// TIA Portal V17 export
// export: Created 2023-02-14T02:49:46.4601409Z, ExportSetting WithDefaults, DisplayName Totally Integrated Automation Portal, DisplayVersion V17, DisplayName TIA Portal Openness, DisplayVersion V17, DisplayName TIA Portal Teamcenter Gateway, DisplayVersion V17, DisplayName TIA Portal Version Control Interface, DisplayVersion V17, DisplayName SINAMICS Startdrive Advanced, DisplayVersion V17, DisplayName SINAMICS Startdrive G130, G150, S120, S150, SINAMICS MV, S210, DisplayVersion V17, DisplayName SINAMICS Startdrive G110M, G120, G120C, G120D, G120P, G115D, DisplayVersion V17, DisplayName STEP 7 Professional, DisplayVersion V17, DisplayName STEP 7 Safety, DisplayVersion V17, DisplayName WinCC Professional, DisplayVersion V17
FUNCTION "IO Homoge" : Void   // FC1, LAD
{ S7_Optimized_Access := 'TRUE' }
VERSION : 0.1
// stored: AutoNumber true, IsIECCheckEnabled false, SetENOAutomatically false, UDAEnableTagReadback false
BEGIN

REGION Network 1: Analog
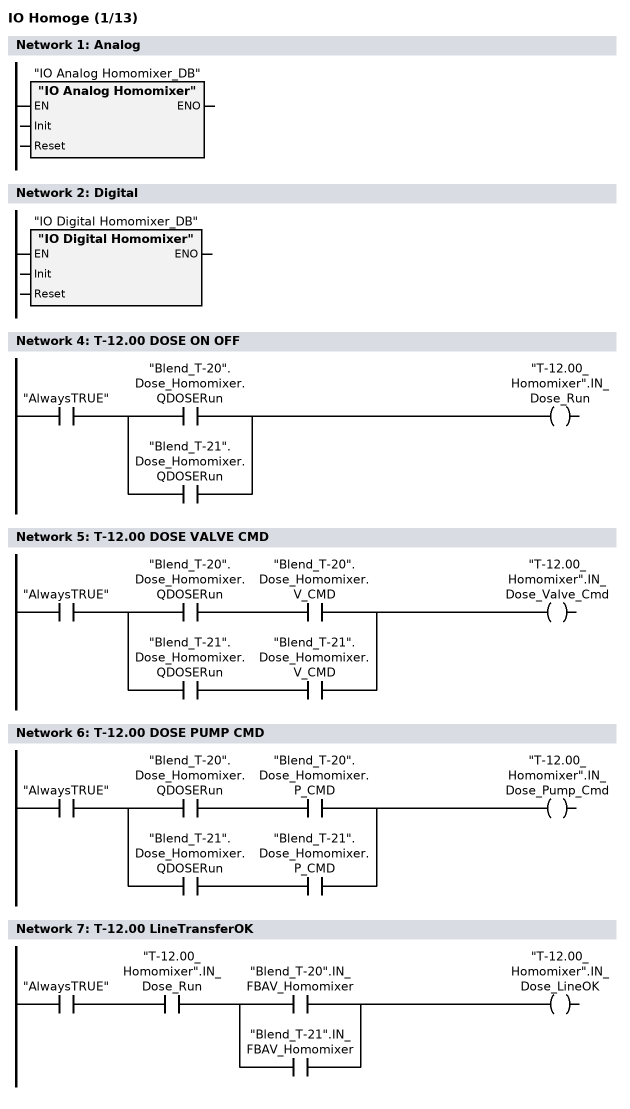
   RUNG wire#powerrail
      "IO Analog Homomixer_DB"(Init :=, Reset :=)
   END_RUNG
   // the same network as SCL:
   "IO Analog Homomixer_DB"();   // "IO Analog Homomixer"
END_REGION

REGION Network 2: Digital
   RUNG wire#powerrail
      "IO Digital Homomixer_DB"(Init :=, Reset :=)
   END_RUNG
   // the same network as SCL:
   "IO Digital Homomixer_DB"();   // "IO Digital Homomixer"
END_REGION

REGION Network 4: T-12.00 DOSE ON OFF
   RUNG wire#powerrail
      Contact( "AlwaysTRUE" )
      wire#w1
      Contact( "Blend_T-20".Dose_Homomixer.QDOSERun )
      wire#w2
      Coil( "T-12.00_Homomixer".IN_Dose_Run )
   END_RUNG
   RUNG wire#w1
      Contact( "Blend_T-21".Dose_Homomixer.QDOSERun )
   END_RUNG wire#w2
   // the same network as SCL:
   "T-12.00_Homomixer".IN_Dose_Run := "AlwaysTRUE" AND ("Blend_T-20".Dose_Homomixer.QDOSERun OR "Blend_T-21".Dose_Homomixer.QDOSERun);
END_REGION

REGION Network 5: T-12.00 DOSE VALVE CMD
   RUNG wire#powerrail
      Contact( "AlwaysTRUE" )
      wire#w1
      Contact( "Blend_T-20".Dose_Homomixer.QDOSERun )
      Contact( "Blend_T-20".Dose_Homomixer.V_CMD )
      wire#w2
      Coil( "T-12.00_Homomixer".IN_Dose_Valve_Cmd )
   END_RUNG
   RUNG wire#w1
      Contact( "Blend_T-21".Dose_Homomixer.QDOSERun )
      Contact( "Blend_T-21".Dose_Homomixer.V_CMD )
   END_RUNG wire#w2
   // the same network as SCL:
   "T-12.00_Homomixer".IN_Dose_Valve_Cmd := "AlwaysTRUE" AND (("Blend_T-20".Dose_Homomixer.QDOSERun AND "Blend_T-20".Dose_Homomixer.V_CMD) OR ("Blend_T-21".Dose_Homomixer.QDOSERun AND "Blend_T-21".Dose_Homomixer.V_CMD));
END_REGION

REGION Network 6: T-12.00 DOSE PUMP CMD
   RUNG wire#powerrail
      Contact( "AlwaysTRUE" )
      wire#w1
      Contact( "Blend_T-20".Dose_Homomixer.QDOSERun )
      Contact( "Blend_T-20".Dose_Homomixer.P_CMD )
      wire#w2
      Coil( "T-12.00_Homomixer".IN_Dose_Pump_Cmd )
   END_RUNG
   RUNG wire#w1
      Contact( "Blend_T-21".Dose_Homomixer.QDOSERun )
      Contact( "Blend_T-21".Dose_Homomixer.P_CMD )
   END_RUNG wire#w2
   // the same network as SCL:
   "T-12.00_Homomixer".IN_Dose_Pump_Cmd := "AlwaysTRUE" AND (("Blend_T-20".Dose_Homomixer.QDOSERun AND "Blend_T-20".Dose_Homomixer.P_CMD) OR ("Blend_T-21".Dose_Homomixer.QDOSERun AND "Blend_T-21".Dose_Homomixer.P_CMD));
END_REGION

REGION Network 7: T-12.00 LineTransferOK
   RUNG wire#powerrail
      Contact( "AlwaysTRUE" )
      Contact( "T-12.00_Homomixer".IN_Dose_Run )
      wire#w1
      Contact( "Blend_T-20".IN_FBAV_Homomixer )
      wire#w2
      Coil( "T-12.00_Homomixer".IN_Dose_LineOK )
   END_RUNG
   RUNG wire#w1
      Contact( "Blend_T-21".IN_FBAV_Homomixer )
   END_RUNG wire#w2
   // the same network as SCL:
   "T-12.00_Homomixer".IN_Dose_LineOK := "AlwaysTRUE" AND "T-12.00_Homomixer".IN_Dose_Run AND ("Blend_T-20".IN_FBAV_Homomixer OR "Blend_T-21".IN_FBAV_Homomixer);
END_REGION

REGION Network 8: T-12.00 Homomixer
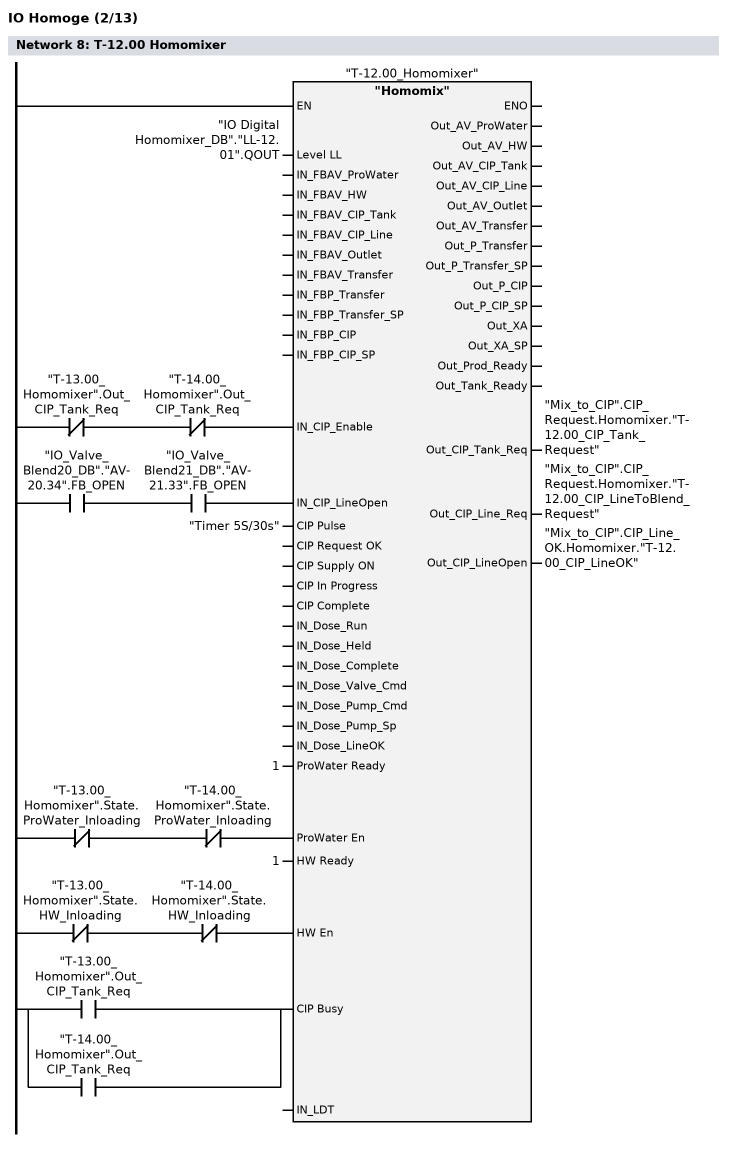
   RUNG wire#powerrail
      "T-12.00_Homomixer"(IN_CIP_Enable := wire#w1, IN_CIP_LineOpen := wire#w2, "ProWater En" := wire#w3, "HW En" := wire#w4, "CIP Busy" := wire#w5, "Level LL" := "IO Digital Homomixer_DB"."LL-12.01".QOUT, IN_FBAV_ProWater :=, IN_FBAV_HW :=, IN_FBAV_CIP_Tank :=, IN_FBAV_CIP_Line :=, IN_FBAV_Outlet :=, IN_FBAV_Transfer :=, IN_FBP_Transfer :=, IN_FBP_Transfer_SP :=, IN_FBP_CIP :=, IN_FBP_CIP_SP :=, "CIP Pulse" := "Timer 5S/30s", "CIP Request OK" :=, "CIP Supply ON" :=, "CIP In Progress" :=, "CIP Complete" :=, IN_Dose_Run :=, IN_Dose_Held :=, IN_Dose_Complete :=, IN_Dose_Valve_Cmd :=, IN_Dose_Pump_Cmd :=, IN_Dose_Pump_Sp :=, IN_Dose_LineOK :=, "ProWater Ready" := 1, "HW Ready" := 1, IN_LDT :=, Out_AV_ProWater =>, Out_AV_HW =>, Out_AV_CIP_Tank =>, Out_AV_CIP_Line =>, Out_AV_Outlet =>, Out_AV_Transfer =>, Out_P_Transfer =>, Out_P_Transfer_SP =>, Out_P_CIP =>, Out_P_CIP_SP =>, Out_XA =>, Out_XA_SP =>, Out_Prod_Ready =>, Out_Tank_Ready =>, Out_CIP_Tank_Req => "Mix_to_CIP".CIP_Request.Homomixer."T-12.00_CIP_Tank_Request", Out_CIP_Line_Req => "Mix_to_CIP".CIP_Request.Homomixer."T-12.00_CIP_LineToBlend_Request", Out_CIP_LineOpen => "Mix_to_CIP".CIP_Line_OK.Homomixer."T-12.00_CIP_LineOK")
   END_RUNG
   RUNG wire#powerrail
      I_Contact( "T-13.00_Homomixer".Out_CIP_Tank_Req )
      I_Contact( "T-14.00_Homomixer".Out_CIP_Tank_Req )
   END_RUNG wire#w1
   RUNG wire#powerrail
      Contact( "IO_Valve_Blend20_DB"."AV-20.34".FB_OPEN )
      Contact( "IO_Valve_Blend21_DB"."AV-21.33".FB_OPEN )
   END_RUNG wire#w2
   RUNG wire#powerrail
      I_Contact( "T-13.00_Homomixer".State.ProWater_Inloading )
      I_Contact( "T-14.00_Homomixer".State.ProWater_Inloading )
   END_RUNG wire#w3
   RUNG wire#powerrail
      I_Contact( "T-13.00_Homomixer".State.HW_Inloading )
      I_Contact( "T-14.00_Homomixer".State.HW_Inloading )
   END_RUNG wire#w4
   RUNG wire#powerrail
      Contact( "T-13.00_Homomixer".Out_CIP_Tank_Req )
   END_RUNG wire#w5
   RUNG wire#powerrail
      Contact( "T-14.00_Homomixer".Out_CIP_Tank_Req )
   END_RUNG wire#w5
   // the same network as SCL:
   "T-12.00_Homomixer"("Level LL" := "IO Digital Homomixer_DB"."LL-12.01".QOUT,   // "Homomix"
                       IN_CIP_Enable := NOT "T-13.00_Homomixer".Out_CIP_Tank_Req AND NOT "T-14.00_Homomixer".Out_CIP_Tank_Req,
                       IN_CIP_LineOpen := "IO_Valve_Blend20_DB"."AV-20.34".FB_OPEN AND "IO_Valve_Blend21_DB"."AV-21.33".FB_OPEN,
                       "CIP Pulse" := "Timer 5S/30s",
                       "ProWater Ready" := 1,
                       "ProWater En" := NOT "T-13.00_Homomixer".State.ProWater_Inloading AND NOT "T-14.00_Homomixer".State.ProWater_Inloading,
                       "HW Ready" := 1,
                       "HW En" := NOT "T-13.00_Homomixer".State.HW_Inloading AND NOT "T-14.00_Homomixer".State.HW_Inloading,
                       "CIP Busy" := "T-13.00_Homomixer".Out_CIP_Tank_Req OR "T-14.00_Homomixer".Out_CIP_Tank_Req,
                       Out_CIP_Tank_Req => "Mix_to_CIP".CIP_Request.Homomixer."T-12.00_CIP_Tank_Request",
                       Out_CIP_Line_Req => "Mix_to_CIP".CIP_Request.Homomixer."T-12.00_CIP_LineToBlend_Request",
                       Out_CIP_LineOpen => "Mix_to_CIP".CIP_Line_OK.Homomixer."T-12.00_CIP_LineOK");
END_REGION

REGION Network 9: T-12.00 Valve Cmd
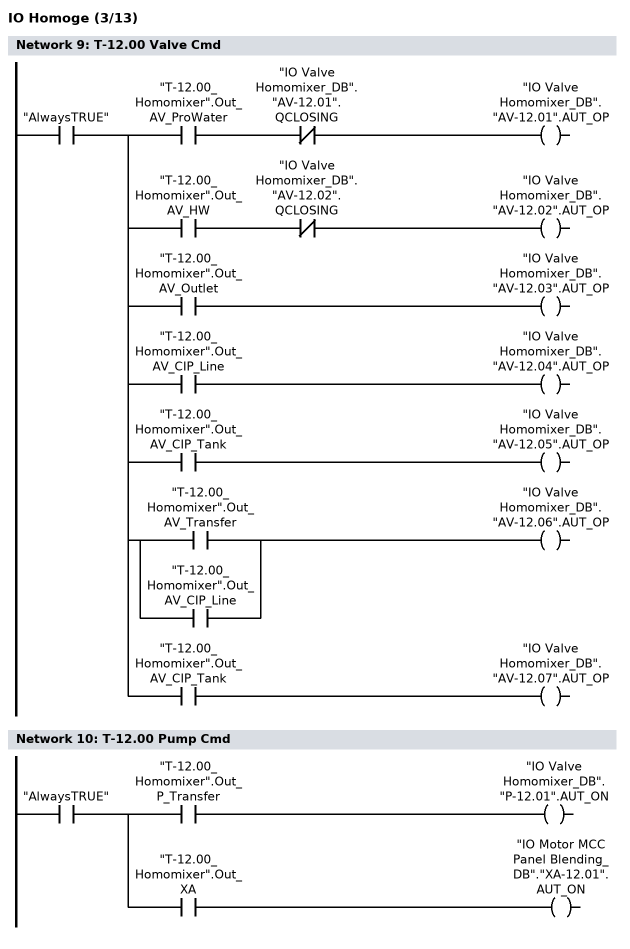
   RUNG wire#powerrail
      Contact( "AlwaysTRUE" )
      wire#w1
      Contact( "T-12.00_Homomixer".Out_AV_ProWater )
      I_Contact( "IO Valve Homomixer_DB"."AV-12.01".QCLOSING )
      Coil( "IO Valve Homomixer_DB"."AV-12.01".AUT_OP )
   END_RUNG
   RUNG wire#w1
      Contact( "T-12.00_Homomixer".Out_AV_HW )
      I_Contact( "IO Valve Homomixer_DB"."AV-12.02".QCLOSING )
      Coil( "IO Valve Homomixer_DB"."AV-12.02".AUT_OP )
   END_RUNG
   RUNG wire#w1
      Contact( "T-12.00_Homomixer".Out_AV_Outlet )
      Coil( "IO Valve Homomixer_DB"."AV-12.03".AUT_OP )
   END_RUNG
   RUNG wire#w1
      Contact( "T-12.00_Homomixer".Out_AV_CIP_Line )
      Coil( "IO Valve Homomixer_DB"."AV-12.04".AUT_OP )
   END_RUNG
   RUNG wire#w1
      Contact( "T-12.00_Homomixer".Out_AV_CIP_Tank )
      Coil( "IO Valve Homomixer_DB"."AV-12.05".AUT_OP )
   END_RUNG
   RUNG wire#w1
      Contact( "T-12.00_Homomixer".Out_AV_Transfer )
      wire#w2
      Coil( "IO Valve Homomixer_DB"."AV-12.06".AUT_OP )
   END_RUNG
   RUNG wire#w1
      Contact( "T-12.00_Homomixer".Out_AV_CIP_Line )
   END_RUNG wire#w2
   RUNG wire#w1
      Contact( "T-12.00_Homomixer".Out_AV_CIP_Tank )
      Coil( "IO Valve Homomixer_DB"."AV-12.07".AUT_OP )
   END_RUNG
   // the same network as SCL:
   "IO Valve Homomixer_DB"."AV-12.01".AUT_OP := "AlwaysTRUE" AND "T-12.00_Homomixer".Out_AV_ProWater AND NOT "IO Valve Homomixer_DB"."AV-12.01".QCLOSING;
   "IO Valve Homomixer_DB"."AV-12.02".AUT_OP := "AlwaysTRUE" AND "T-12.00_Homomixer".Out_AV_HW AND NOT "IO Valve Homomixer_DB"."AV-12.02".QCLOSING;
   "IO Valve Homomixer_DB"."AV-12.03".AUT_OP := "AlwaysTRUE" AND "T-12.00_Homomixer".Out_AV_Outlet;
   "IO Valve Homomixer_DB"."AV-12.04".AUT_OP := "AlwaysTRUE" AND "T-12.00_Homomixer".Out_AV_CIP_Line;
   "IO Valve Homomixer_DB"."AV-12.05".AUT_OP := "AlwaysTRUE" AND "T-12.00_Homomixer".Out_AV_CIP_Tank;
   "IO Valve Homomixer_DB"."AV-12.06".AUT_OP := "AlwaysTRUE" AND ("T-12.00_Homomixer".Out_AV_Transfer OR "T-12.00_Homomixer".Out_AV_CIP_Line);
   "IO Valve Homomixer_DB"."AV-12.07".AUT_OP := "AlwaysTRUE" AND "T-12.00_Homomixer".Out_AV_CIP_Tank;
END_REGION

REGION Network 10: T-12.00 Pump Cmd
   RUNG wire#powerrail
      Contact( "AlwaysTRUE" )
      wire#w1
      Contact( "T-12.00_Homomixer".Out_P_Transfer )
      Coil( "IO Valve Homomixer_DB"."P-12.01".AUT_ON )
   END_RUNG
   RUNG wire#w1
      Contact( "T-12.00_Homomixer".Out_XA )
      Coil( "IO Motor MCC Panel Blending_DB"."XA-12.01".AUT_ON )
   END_RUNG
   // the same network as SCL:
   "IO Valve Homomixer_DB"."P-12.01".AUT_ON := "AlwaysTRUE" AND "T-12.00_Homomixer".Out_P_Transfer;
   "IO Motor MCC Panel Blending_DB"."XA-12.01".AUT_ON := "AlwaysTRUE" AND "T-12.00_Homomixer".Out_XA;
END_REGION

REGION Network 11: T-12.00 Feedback Instrument
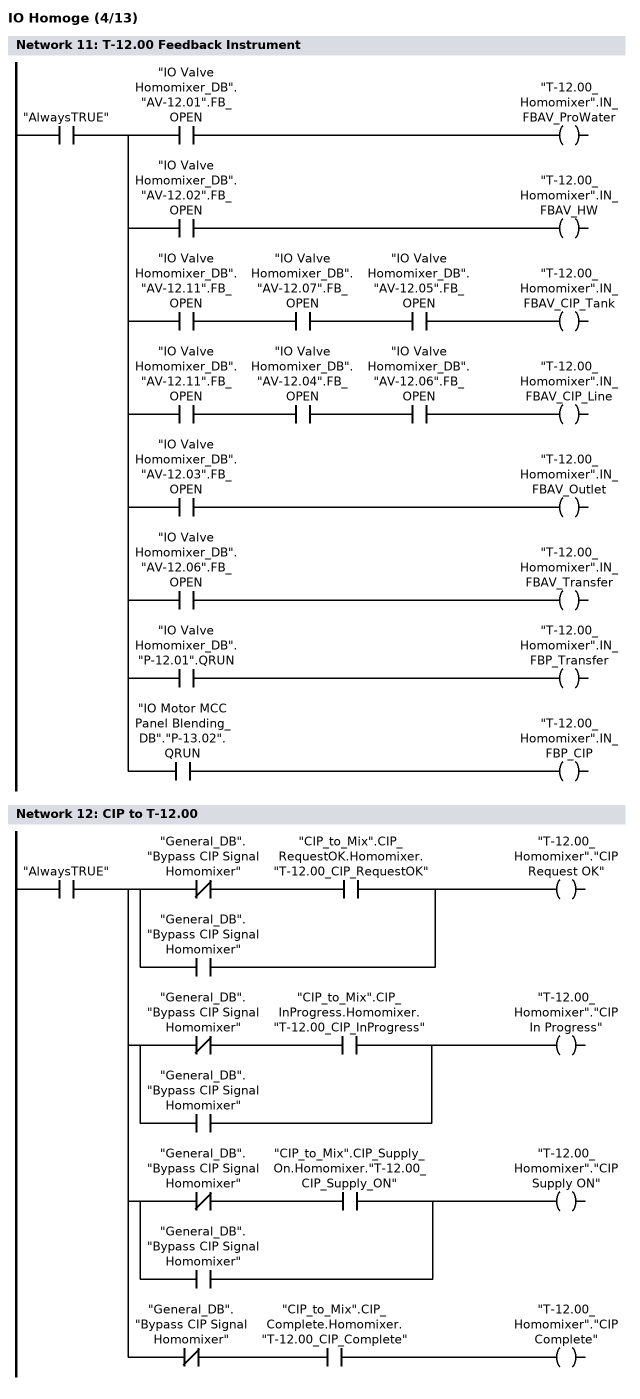
   RUNG wire#powerrail
      Contact( "AlwaysTRUE" )
      wire#w1
      Contact( "IO Valve Homomixer_DB"."AV-12.01".FB_OPEN )
      Coil( "T-12.00_Homomixer".IN_FBAV_ProWater )
   END_RUNG
   RUNG wire#w1
      Contact( "IO Valve Homomixer_DB"."AV-12.02".FB_OPEN )
      Coil( "T-12.00_Homomixer".IN_FBAV_HW )
   END_RUNG
   RUNG wire#w1
      Contact( "IO Valve Homomixer_DB"."AV-12.11".FB_OPEN )
      Contact( "IO Valve Homomixer_DB"."AV-12.07".FB_OPEN )
      Contact( "IO Valve Homomixer_DB"."AV-12.05".FB_OPEN )
      Coil( "T-12.00_Homomixer".IN_FBAV_CIP_Tank )
   END_RUNG
   RUNG wire#w1
      Contact( "IO Valve Homomixer_DB"."AV-12.11".FB_OPEN )
      Contact( "IO Valve Homomixer_DB"."AV-12.04".FB_OPEN )
      Contact( "IO Valve Homomixer_DB"."AV-12.06".FB_OPEN )
      Coil( "T-12.00_Homomixer".IN_FBAV_CIP_Line )
   END_RUNG
   RUNG wire#w1
      Contact( "IO Valve Homomixer_DB"."AV-12.03".FB_OPEN )
      Coil( "T-12.00_Homomixer".IN_FBAV_Outlet )
   END_RUNG
   RUNG wire#w1
      Contact( "IO Valve Homomixer_DB"."AV-12.06".FB_OPEN )
      Coil( "T-12.00_Homomixer".IN_FBAV_Transfer )
   END_RUNG
   RUNG wire#w1
      Contact( "IO Valve Homomixer_DB"."P-12.01".QRUN )
      Coil( "T-12.00_Homomixer".IN_FBP_Transfer )
   END_RUNG
   RUNG wire#w1
      Contact( "IO Motor MCC Panel Blending_DB"."P-13.02".QRUN )
      Coil( "T-12.00_Homomixer".IN_FBP_CIP )
   END_RUNG
   // the same network as SCL:
   "T-12.00_Homomixer".IN_FBAV_ProWater := "AlwaysTRUE" AND "IO Valve Homomixer_DB"."AV-12.01".FB_OPEN;
   "T-12.00_Homomixer".IN_FBAV_HW := "AlwaysTRUE" AND "IO Valve Homomixer_DB"."AV-12.02".FB_OPEN;
   "T-12.00_Homomixer".IN_FBAV_CIP_Tank := "AlwaysTRUE" AND "IO Valve Homomixer_DB"."AV-12.11".FB_OPEN AND "IO Valve Homomixer_DB"."AV-12.07".FB_OPEN AND "IO Valve Homomixer_DB"."AV-12.05".FB_OPEN;
   "T-12.00_Homomixer".IN_FBAV_CIP_Line := "AlwaysTRUE" AND "IO Valve Homomixer_DB"."AV-12.11".FB_OPEN AND "IO Valve Homomixer_DB"."AV-12.04".FB_OPEN AND "IO Valve Homomixer_DB"."AV-12.06".FB_OPEN;
   "T-12.00_Homomixer".IN_FBAV_Outlet := "AlwaysTRUE" AND "IO Valve Homomixer_DB"."AV-12.03".FB_OPEN;
   "T-12.00_Homomixer".IN_FBAV_Transfer := "AlwaysTRUE" AND "IO Valve Homomixer_DB"."AV-12.06".FB_OPEN;
   "T-12.00_Homomixer".IN_FBP_Transfer := "AlwaysTRUE" AND "IO Valve Homomixer_DB"."P-12.01".QRUN;
   "T-12.00_Homomixer".IN_FBP_CIP := "AlwaysTRUE" AND "IO Motor MCC Panel Blending_DB"."P-13.02".QRUN;
END_REGION

REGION Network 12: CIP to T-12.00
   RUNG wire#powerrail
      Contact( "AlwaysTRUE" )
      wire#w1
      I_Contact( "General_DB"."Bypass CIP Signal Homomixer" )
      Contact( "CIP_to_Mix".CIP_RequestOK.Homomixer."T-12.00_CIP_RequestOK" )
      wire#w2
      Coil( "T-12.00_Homomixer"."CIP Request OK" )
   END_RUNG
   RUNG wire#w1
      Contact( "General_DB"."Bypass CIP Signal Homomixer" )
   END_RUNG wire#w2
   RUNG wire#w1
      I_Contact( "General_DB"."Bypass CIP Signal Homomixer" )
      Contact( "CIP_to_Mix".CIP_InProgress.Homomixer."T-12.00_CIP_InProgress" )
      wire#w3
      Coil( "T-12.00_Homomixer"."CIP In Progress" )
   END_RUNG
   RUNG wire#w1
      Contact( "General_DB"."Bypass CIP Signal Homomixer" )
   END_RUNG wire#w3
   RUNG wire#w1
      I_Contact( "General_DB"."Bypass CIP Signal Homomixer" )
      Contact( "CIP_to_Mix".CIP_Supply_On.Homomixer."T-12.00_CIP_Supply_ON" )
      wire#w4
      Coil( "T-12.00_Homomixer"."CIP Supply ON" )
   END_RUNG
   RUNG wire#w1
      Contact( "General_DB"."Bypass CIP Signal Homomixer" )
   END_RUNG wire#w4
   RUNG wire#w1
      I_Contact( "General_DB"."Bypass CIP Signal Homomixer" )
      Contact( "CIP_to_Mix".CIP_Complete.Homomixer."T-12.00_CIP_Complete" )
      Coil( "T-12.00_Homomixer"."CIP Complete" )
   END_RUNG
   // the same network as SCL:
   "T-12.00_Homomixer"."CIP Request OK" := "AlwaysTRUE" AND ((NOT "General_DB"."Bypass CIP Signal Homomixer" AND "CIP_to_Mix".CIP_RequestOK.Homomixer."T-12.00_CIP_RequestOK") OR "General_DB"."Bypass CIP Signal Homomixer");
   "T-12.00_Homomixer"."CIP In Progress" := "AlwaysTRUE" AND ((NOT "General_DB"."Bypass CIP Signal Homomixer" AND "CIP_to_Mix".CIP_InProgress.Homomixer."T-12.00_CIP_InProgress") OR "General_DB"."Bypass CIP Signal Homomixer");
   "T-12.00_Homomixer"."CIP Supply ON" := "AlwaysTRUE" AND ((NOT "General_DB"."Bypass CIP Signal Homomixer" AND "CIP_to_Mix".CIP_Supply_On.Homomixer."T-12.00_CIP_Supply_ON") OR "General_DB"."Bypass CIP Signal Homomixer");
   "T-12.00_Homomixer"."CIP Complete" := "AlwaysTRUE" AND NOT "General_DB"."Bypass CIP Signal Homomixer" AND "CIP_to_Mix".CIP_Complete.Homomixer."T-12.00_CIP_Complete";
END_REGION

REGION Network 15: T-13.00 DOSE ON OFF
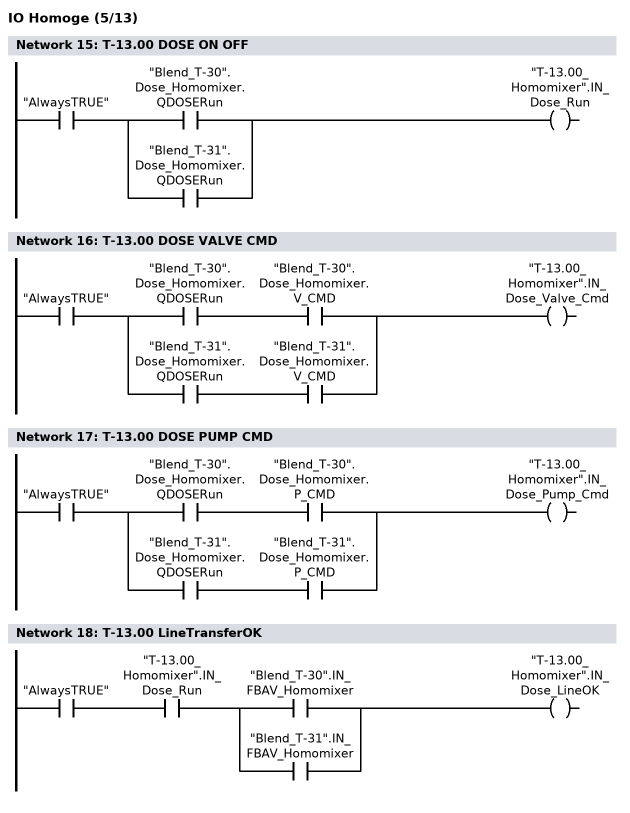
   RUNG wire#powerrail
      Contact( "AlwaysTRUE" )
      wire#w1
      Contact( "Blend_T-30".Dose_Homomixer.QDOSERun )
      wire#w2
      Coil( "T-13.00_Homomixer".IN_Dose_Run )
   END_RUNG
   RUNG wire#w1
      Contact( "Blend_T-31".Dose_Homomixer.QDOSERun )
   END_RUNG wire#w2
   // the same network as SCL:
   "T-13.00_Homomixer".IN_Dose_Run := "AlwaysTRUE" AND ("Blend_T-30".Dose_Homomixer.QDOSERun OR "Blend_T-31".Dose_Homomixer.QDOSERun);
END_REGION

REGION Network 16: T-13.00 DOSE VALVE CMD
   RUNG wire#powerrail
      Contact( "AlwaysTRUE" )
      wire#w1
      Contact( "Blend_T-30".Dose_Homomixer.QDOSERun )
      Contact( "Blend_T-30".Dose_Homomixer.V_CMD )
      wire#w2
      Coil( "T-13.00_Homomixer".IN_Dose_Valve_Cmd )
   END_RUNG
   RUNG wire#w1
      Contact( "Blend_T-31".Dose_Homomixer.QDOSERun )
      Contact( "Blend_T-31".Dose_Homomixer.V_CMD )
   END_RUNG wire#w2
   // the same network as SCL:
   "T-13.00_Homomixer".IN_Dose_Valve_Cmd := "AlwaysTRUE" AND (("Blend_T-30".Dose_Homomixer.QDOSERun AND "Blend_T-30".Dose_Homomixer.V_CMD) OR ("Blend_T-31".Dose_Homomixer.QDOSERun AND "Blend_T-31".Dose_Homomixer.V_CMD));
END_REGION

REGION Network 17: T-13.00 DOSE PUMP CMD
   RUNG wire#powerrail
      Contact( "AlwaysTRUE" )
      wire#w1
      Contact( "Blend_T-30".Dose_Homomixer.QDOSERun )
      Contact( "Blend_T-30".Dose_Homomixer.P_CMD )
      wire#w2
      Coil( "T-13.00_Homomixer".IN_Dose_Pump_Cmd )
   END_RUNG
   RUNG wire#w1
      Contact( "Blend_T-31".Dose_Homomixer.QDOSERun )
      Contact( "Blend_T-31".Dose_Homomixer.P_CMD )
   END_RUNG wire#w2
   // the same network as SCL:
   "T-13.00_Homomixer".IN_Dose_Pump_Cmd := "AlwaysTRUE" AND (("Blend_T-30".Dose_Homomixer.QDOSERun AND "Blend_T-30".Dose_Homomixer.P_CMD) OR ("Blend_T-31".Dose_Homomixer.QDOSERun AND "Blend_T-31".Dose_Homomixer.P_CMD));
END_REGION

REGION Network 18: T-13.00 LineTransferOK
   RUNG wire#powerrail
      Contact( "AlwaysTRUE" )
      Contact( "T-13.00_Homomixer".IN_Dose_Run )
      wire#w1
      Contact( "Blend_T-30".IN_FBAV_Homomixer )
      wire#w2
      Coil( "T-13.00_Homomixer".IN_Dose_LineOK )
   END_RUNG
   RUNG wire#w1
      Contact( "Blend_T-31".IN_FBAV_Homomixer )
   END_RUNG wire#w2
   // the same network as SCL:
   "T-13.00_Homomixer".IN_Dose_LineOK := "AlwaysTRUE" AND "T-13.00_Homomixer".IN_Dose_Run AND ("Blend_T-30".IN_FBAV_Homomixer OR "Blend_T-31".IN_FBAV_Homomixer);
END_REGION

REGION Network 19: T-13.00 Homomixer
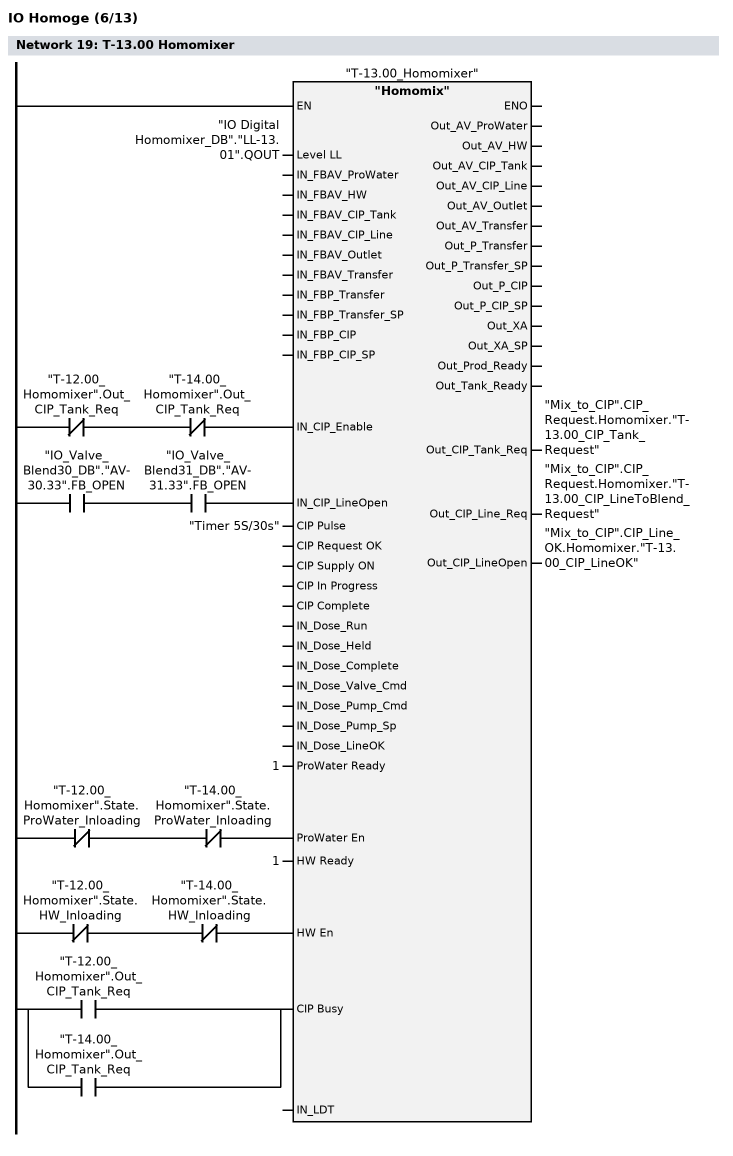
   RUNG wire#powerrail
      "T-13.00_Homomixer"(IN_CIP_Enable := wire#w1, IN_CIP_LineOpen := wire#w2, "ProWater En" := wire#w3, "HW En" := wire#w4, "CIP Busy" := wire#w5, "Level LL" := "IO Digital Homomixer_DB"."LL-13.01".QOUT, IN_FBAV_ProWater :=, IN_FBAV_HW :=, IN_FBAV_CIP_Tank :=, IN_FBAV_CIP_Line :=, IN_FBAV_Outlet :=, IN_FBAV_Transfer :=, IN_FBP_Transfer :=, IN_FBP_Transfer_SP :=, IN_FBP_CIP :=, IN_FBP_CIP_SP :=, "CIP Pulse" := "Timer 5S/30s", "CIP Request OK" :=, "CIP Supply ON" :=, "CIP In Progress" :=, "CIP Complete" :=, IN_Dose_Run :=, IN_Dose_Held :=, IN_Dose_Complete :=, IN_Dose_Valve_Cmd :=, IN_Dose_Pump_Cmd :=, IN_Dose_Pump_Sp :=, IN_Dose_LineOK :=, "ProWater Ready" := 1, "HW Ready" := 1, IN_LDT :=, Out_AV_ProWater =>, Out_AV_HW =>, Out_AV_CIP_Tank =>, Out_AV_CIP_Line =>, Out_AV_Outlet =>, Out_AV_Transfer =>, Out_P_Transfer =>, Out_P_Transfer_SP =>, Out_P_CIP =>, Out_P_CIP_SP =>, Out_XA =>, Out_XA_SP =>, Out_Prod_Ready =>, Out_Tank_Ready =>, Out_CIP_Tank_Req => "Mix_to_CIP".CIP_Request.Homomixer."T-13.00_CIP_Tank_Request", Out_CIP_Line_Req => "Mix_to_CIP".CIP_Request.Homomixer."T-13.00_CIP_LineToBlend_Request", Out_CIP_LineOpen => "Mix_to_CIP".CIP_Line_OK.Homomixer."T-13.00_CIP_LineOK")
   END_RUNG
   RUNG wire#powerrail
      I_Contact( "T-12.00_Homomixer".Out_CIP_Tank_Req )
      I_Contact( "T-14.00_Homomixer".Out_CIP_Tank_Req )
   END_RUNG wire#w1
   RUNG wire#powerrail
      Contact( "IO_Valve_Blend30_DB"."AV-30.33".FB_OPEN )
      Contact( "IO_Valve_Blend31_DB"."AV-31.33".FB_OPEN )
   END_RUNG wire#w2
   RUNG wire#powerrail
      I_Contact( "T-12.00_Homomixer".State.ProWater_Inloading )
      I_Contact( "T-14.00_Homomixer".State.ProWater_Inloading )
   END_RUNG wire#w3
   RUNG wire#powerrail
      I_Contact( "T-12.00_Homomixer".State.HW_Inloading )
      I_Contact( "T-14.00_Homomixer".State.HW_Inloading )
   END_RUNG wire#w4
   RUNG wire#powerrail
      Contact( "T-12.00_Homomixer".Out_CIP_Tank_Req )
   END_RUNG wire#w5
   RUNG wire#powerrail
      Contact( "T-14.00_Homomixer".Out_CIP_Tank_Req )
   END_RUNG wire#w5
   // the same network as SCL:
   "T-13.00_Homomixer"("Level LL" := "IO Digital Homomixer_DB"."LL-13.01".QOUT,   // "Homomix"
                       IN_CIP_Enable := NOT "T-12.00_Homomixer".Out_CIP_Tank_Req AND NOT "T-14.00_Homomixer".Out_CIP_Tank_Req,
                       IN_CIP_LineOpen := "IO_Valve_Blend30_DB"."AV-30.33".FB_OPEN AND "IO_Valve_Blend31_DB"."AV-31.33".FB_OPEN,
                       "CIP Pulse" := "Timer 5S/30s",
                       "ProWater Ready" := 1,
                       "ProWater En" := NOT "T-12.00_Homomixer".State.ProWater_Inloading AND NOT "T-14.00_Homomixer".State.ProWater_Inloading,
                       "HW Ready" := 1,
                       "HW En" := NOT "T-12.00_Homomixer".State.HW_Inloading AND NOT "T-14.00_Homomixer".State.HW_Inloading,
                       "CIP Busy" := "T-12.00_Homomixer".Out_CIP_Tank_Req OR "T-14.00_Homomixer".Out_CIP_Tank_Req,
                       Out_CIP_Tank_Req => "Mix_to_CIP".CIP_Request.Homomixer."T-13.00_CIP_Tank_Request",
                       Out_CIP_Line_Req => "Mix_to_CIP".CIP_Request.Homomixer."T-13.00_CIP_LineToBlend_Request",
                       Out_CIP_LineOpen => "Mix_to_CIP".CIP_Line_OK.Homomixer."T-13.00_CIP_LineOK");
END_REGION

REGION Network 20: T-13.00 Valve Cmd
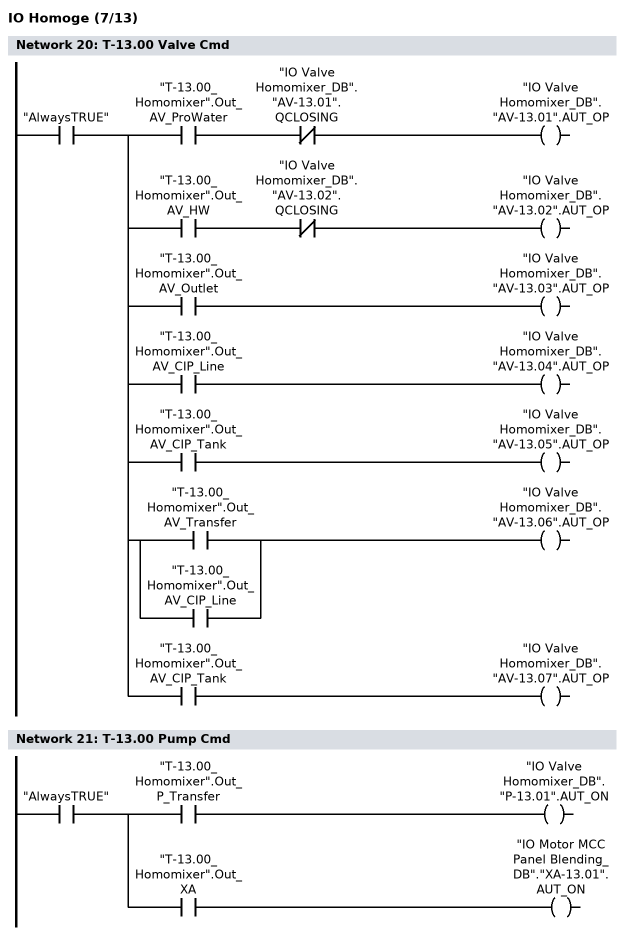
   RUNG wire#powerrail
      Contact( "AlwaysTRUE" )
      wire#w1
      Contact( "T-13.00_Homomixer".Out_AV_ProWater )
      I_Contact( "IO Valve Homomixer_DB"."AV-13.01".QCLOSING )
      Coil( "IO Valve Homomixer_DB"."AV-13.01".AUT_OP )
   END_RUNG
   RUNG wire#w1
      Contact( "T-13.00_Homomixer".Out_AV_HW )
      I_Contact( "IO Valve Homomixer_DB"."AV-13.02".QCLOSING )
      Coil( "IO Valve Homomixer_DB"."AV-13.02".AUT_OP )
   END_RUNG
   RUNG wire#w1
      Contact( "T-13.00_Homomixer".Out_AV_Outlet )
      Coil( "IO Valve Homomixer_DB"."AV-13.03".AUT_OP )
   END_RUNG
   RUNG wire#w1
      Contact( "T-13.00_Homomixer".Out_AV_CIP_Line )
      Coil( "IO Valve Homomixer_DB"."AV-13.04".AUT_OP )
   END_RUNG
   RUNG wire#w1
      Contact( "T-13.00_Homomixer".Out_AV_CIP_Tank )
      Coil( "IO Valve Homomixer_DB"."AV-13.05".AUT_OP )
   END_RUNG
   RUNG wire#w1
      Contact( "T-13.00_Homomixer".Out_AV_Transfer )
      wire#w2
      Coil( "IO Valve Homomixer_DB"."AV-13.06".AUT_OP )
   END_RUNG
   RUNG wire#w1
      Contact( "T-13.00_Homomixer".Out_AV_CIP_Line )
   END_RUNG wire#w2
   RUNG wire#w1
      Contact( "T-13.00_Homomixer".Out_AV_CIP_Tank )
      Coil( "IO Valve Homomixer_DB"."AV-13.07".AUT_OP )
   END_RUNG
   // the same network as SCL:
   "IO Valve Homomixer_DB"."AV-13.01".AUT_OP := "AlwaysTRUE" AND "T-13.00_Homomixer".Out_AV_ProWater AND NOT "IO Valve Homomixer_DB"."AV-13.01".QCLOSING;
   "IO Valve Homomixer_DB"."AV-13.02".AUT_OP := "AlwaysTRUE" AND "T-13.00_Homomixer".Out_AV_HW AND NOT "IO Valve Homomixer_DB"."AV-13.02".QCLOSING;
   "IO Valve Homomixer_DB"."AV-13.03".AUT_OP := "AlwaysTRUE" AND "T-13.00_Homomixer".Out_AV_Outlet;
   "IO Valve Homomixer_DB"."AV-13.04".AUT_OP := "AlwaysTRUE" AND "T-13.00_Homomixer".Out_AV_CIP_Line;
   "IO Valve Homomixer_DB"."AV-13.05".AUT_OP := "AlwaysTRUE" AND "T-13.00_Homomixer".Out_AV_CIP_Tank;
   "IO Valve Homomixer_DB"."AV-13.06".AUT_OP := "AlwaysTRUE" AND ("T-13.00_Homomixer".Out_AV_Transfer OR "T-13.00_Homomixer".Out_AV_CIP_Line);
   "IO Valve Homomixer_DB"."AV-13.07".AUT_OP := "AlwaysTRUE" AND "T-13.00_Homomixer".Out_AV_CIP_Tank;
END_REGION

REGION Network 21: T-13.00 Pump Cmd
   RUNG wire#powerrail
      Contact( "AlwaysTRUE" )
      wire#w1
      Contact( "T-13.00_Homomixer".Out_P_Transfer )
      Coil( "IO Valve Homomixer_DB"."P-13.01".AUT_ON )
   END_RUNG
   RUNG wire#w1
      Contact( "T-13.00_Homomixer".Out_XA )
      Coil( "IO Motor MCC Panel Blending_DB"."XA-13.01".AUT_ON )
   END_RUNG
   // the same network as SCL:
   "IO Valve Homomixer_DB"."P-13.01".AUT_ON := "AlwaysTRUE" AND "T-13.00_Homomixer".Out_P_Transfer;
   "IO Motor MCC Panel Blending_DB"."XA-13.01".AUT_ON := "AlwaysTRUE" AND "T-13.00_Homomixer".Out_XA;
END_REGION

REGION Network 22: T-13.00 Feedback Instrument
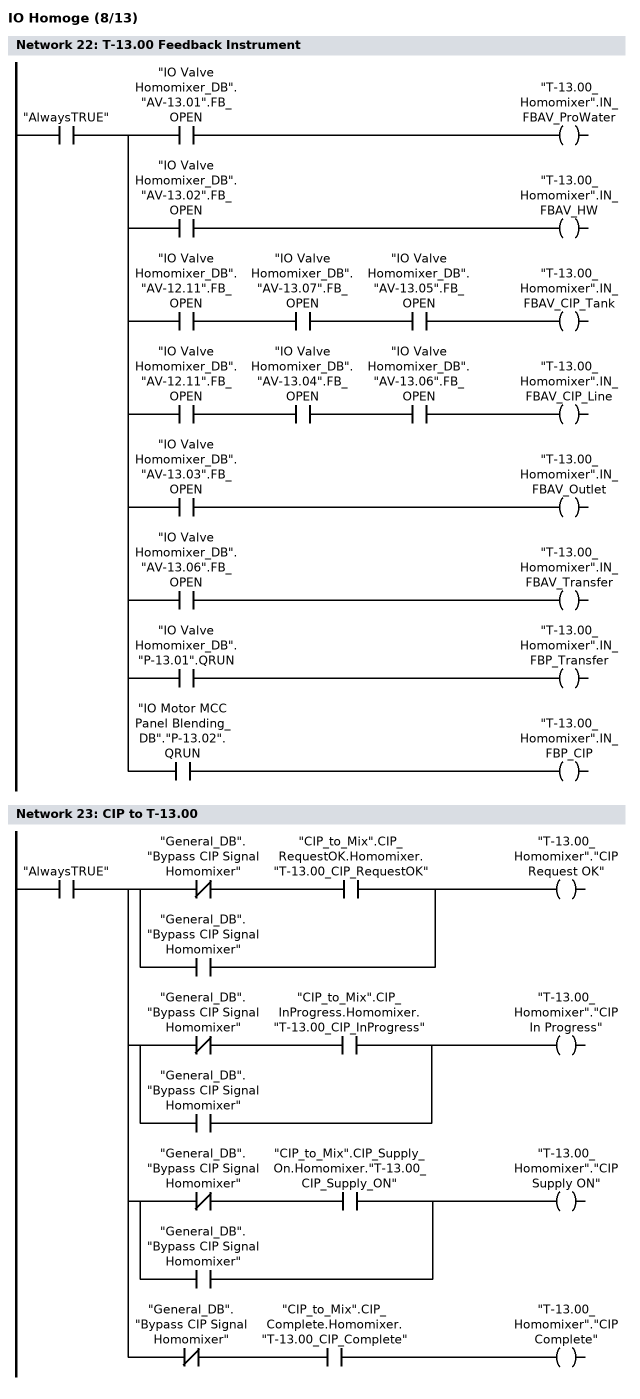
   RUNG wire#powerrail
      Contact( "AlwaysTRUE" )
      wire#w1
      Contact( "IO Valve Homomixer_DB"."AV-13.01".FB_OPEN )
      Coil( "T-13.00_Homomixer".IN_FBAV_ProWater )
   END_RUNG
   RUNG wire#w1
      Contact( "IO Valve Homomixer_DB"."AV-13.02".FB_OPEN )
      Coil( "T-13.00_Homomixer".IN_FBAV_HW )
   END_RUNG
   RUNG wire#w1
      Contact( "IO Valve Homomixer_DB"."AV-12.11".FB_OPEN )
      Contact( "IO Valve Homomixer_DB"."AV-13.07".FB_OPEN )
      Contact( "IO Valve Homomixer_DB"."AV-13.05".FB_OPEN )
      Coil( "T-13.00_Homomixer".IN_FBAV_CIP_Tank )
   END_RUNG
   RUNG wire#w1
      Contact( "IO Valve Homomixer_DB"."AV-12.11".FB_OPEN )
      Contact( "IO Valve Homomixer_DB"."AV-13.04".FB_OPEN )
      Contact( "IO Valve Homomixer_DB"."AV-13.06".FB_OPEN )
      Coil( "T-13.00_Homomixer".IN_FBAV_CIP_Line )
   END_RUNG
   RUNG wire#w1
      Contact( "IO Valve Homomixer_DB"."AV-13.03".FB_OPEN )
      Coil( "T-13.00_Homomixer".IN_FBAV_Outlet )
   END_RUNG
   RUNG wire#w1
      Contact( "IO Valve Homomixer_DB"."AV-13.06".FB_OPEN )
      Coil( "T-13.00_Homomixer".IN_FBAV_Transfer )
   END_RUNG
   RUNG wire#w1
      Contact( "IO Valve Homomixer_DB"."P-13.01".QRUN )
      Coil( "T-13.00_Homomixer".IN_FBP_Transfer )
   END_RUNG
   RUNG wire#w1
      Contact( "IO Motor MCC Panel Blending_DB"."P-13.02".QRUN )
      Coil( "T-13.00_Homomixer".IN_FBP_CIP )
   END_RUNG
   // the same network as SCL:
   "T-13.00_Homomixer".IN_FBAV_ProWater := "AlwaysTRUE" AND "IO Valve Homomixer_DB"."AV-13.01".FB_OPEN;
   "T-13.00_Homomixer".IN_FBAV_HW := "AlwaysTRUE" AND "IO Valve Homomixer_DB"."AV-13.02".FB_OPEN;
   "T-13.00_Homomixer".IN_FBAV_CIP_Tank := "AlwaysTRUE" AND "IO Valve Homomixer_DB"."AV-12.11".FB_OPEN AND "IO Valve Homomixer_DB"."AV-13.07".FB_OPEN AND "IO Valve Homomixer_DB"."AV-13.05".FB_OPEN;
   "T-13.00_Homomixer".IN_FBAV_CIP_Line := "AlwaysTRUE" AND "IO Valve Homomixer_DB"."AV-12.11".FB_OPEN AND "IO Valve Homomixer_DB"."AV-13.04".FB_OPEN AND "IO Valve Homomixer_DB"."AV-13.06".FB_OPEN;
   "T-13.00_Homomixer".IN_FBAV_Outlet := "AlwaysTRUE" AND "IO Valve Homomixer_DB"."AV-13.03".FB_OPEN;
   "T-13.00_Homomixer".IN_FBAV_Transfer := "AlwaysTRUE" AND "IO Valve Homomixer_DB"."AV-13.06".FB_OPEN;
   "T-13.00_Homomixer".IN_FBP_Transfer := "AlwaysTRUE" AND "IO Valve Homomixer_DB"."P-13.01".QRUN;
   "T-13.00_Homomixer".IN_FBP_CIP := "AlwaysTRUE" AND "IO Motor MCC Panel Blending_DB"."P-13.02".QRUN;
END_REGION

REGION Network 23: CIP to T-13.00
   RUNG wire#powerrail
      Contact( "AlwaysTRUE" )
      wire#w1
      I_Contact( "General_DB"."Bypass CIP Signal Homomixer" )
      Contact( "CIP_to_Mix".CIP_RequestOK.Homomixer."T-13.00_CIP_RequestOK" )
      wire#w2
      Coil( "T-13.00_Homomixer"."CIP Request OK" )
   END_RUNG
   RUNG wire#w1
      Contact( "General_DB"."Bypass CIP Signal Homomixer" )
   END_RUNG wire#w2
   RUNG wire#w1
      I_Contact( "General_DB"."Bypass CIP Signal Homomixer" )
      Contact( "CIP_to_Mix".CIP_InProgress.Homomixer."T-13.00_CIP_InProgress" )
      wire#w3
      Coil( "T-13.00_Homomixer"."CIP In Progress" )
   END_RUNG
   RUNG wire#w1
      Contact( "General_DB"."Bypass CIP Signal Homomixer" )
   END_RUNG wire#w3
   RUNG wire#w1
      I_Contact( "General_DB"."Bypass CIP Signal Homomixer" )
      Contact( "CIP_to_Mix".CIP_Supply_On.Homomixer."T-13.00_CIP_Supply_ON" )
      wire#w4
      Coil( "T-13.00_Homomixer"."CIP Supply ON" )
   END_RUNG
   RUNG wire#w1
      Contact( "General_DB"."Bypass CIP Signal Homomixer" )
   END_RUNG wire#w4
   RUNG wire#w1
      I_Contact( "General_DB"."Bypass CIP Signal Homomixer" )
      Contact( "CIP_to_Mix".CIP_Complete.Homomixer."T-13.00_CIP_Complete" )
      Coil( "T-13.00_Homomixer"."CIP Complete" )
   END_RUNG
   // the same network as SCL:
   "T-13.00_Homomixer"."CIP Request OK" := "AlwaysTRUE" AND ((NOT "General_DB"."Bypass CIP Signal Homomixer" AND "CIP_to_Mix".CIP_RequestOK.Homomixer."T-13.00_CIP_RequestOK") OR "General_DB"."Bypass CIP Signal Homomixer");
   "T-13.00_Homomixer"."CIP In Progress" := "AlwaysTRUE" AND ((NOT "General_DB"."Bypass CIP Signal Homomixer" AND "CIP_to_Mix".CIP_InProgress.Homomixer."T-13.00_CIP_InProgress") OR "General_DB"."Bypass CIP Signal Homomixer");
   "T-13.00_Homomixer"."CIP Supply ON" := "AlwaysTRUE" AND ((NOT "General_DB"."Bypass CIP Signal Homomixer" AND "CIP_to_Mix".CIP_Supply_On.Homomixer."T-13.00_CIP_Supply_ON") OR "General_DB"."Bypass CIP Signal Homomixer");
   "T-13.00_Homomixer"."CIP Complete" := "AlwaysTRUE" AND NOT "General_DB"."Bypass CIP Signal Homomixer" AND "CIP_to_Mix".CIP_Complete.Homomixer."T-13.00_CIP_Complete";
END_REGION

REGION Network 26: T-14.00 DOSE ON OFF
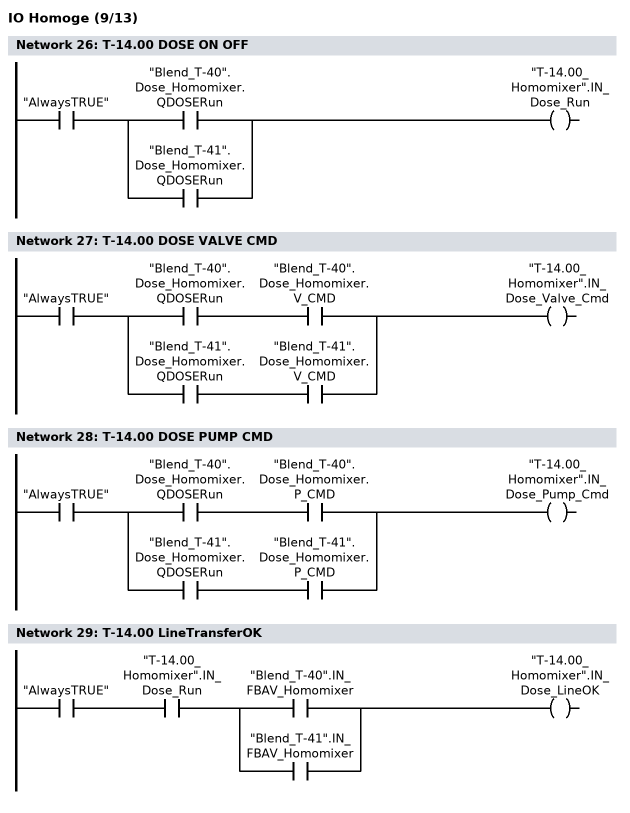
   RUNG wire#powerrail
      Contact( "AlwaysTRUE" )
      wire#w1
      Contact( "Blend_T-40".Dose_Homomixer.QDOSERun )
      wire#w2
      Coil( "T-14.00_Homomixer".IN_Dose_Run )
   END_RUNG
   RUNG wire#w1
      Contact( "Blend_T-41".Dose_Homomixer.QDOSERun )
   END_RUNG wire#w2
   // the same network as SCL:
   "T-14.00_Homomixer".IN_Dose_Run := "AlwaysTRUE" AND ("Blend_T-40".Dose_Homomixer.QDOSERun OR "Blend_T-41".Dose_Homomixer.QDOSERun);
END_REGION

REGION Network 27: T-14.00 DOSE VALVE CMD
   RUNG wire#powerrail
      Contact( "AlwaysTRUE" )
      wire#w1
      Contact( "Blend_T-40".Dose_Homomixer.QDOSERun )
      Contact( "Blend_T-40".Dose_Homomixer.V_CMD )
      wire#w2
      Coil( "T-14.00_Homomixer".IN_Dose_Valve_Cmd )
   END_RUNG
   RUNG wire#w1
      Contact( "Blend_T-41".Dose_Homomixer.QDOSERun )
      Contact( "Blend_T-41".Dose_Homomixer.V_CMD )
   END_RUNG wire#w2
   // the same network as SCL:
   "T-14.00_Homomixer".IN_Dose_Valve_Cmd := "AlwaysTRUE" AND (("Blend_T-40".Dose_Homomixer.QDOSERun AND "Blend_T-40".Dose_Homomixer.V_CMD) OR ("Blend_T-41".Dose_Homomixer.QDOSERun AND "Blend_T-41".Dose_Homomixer.V_CMD));
END_REGION

REGION Network 28: T-14.00 DOSE PUMP CMD
   RUNG wire#powerrail
      Contact( "AlwaysTRUE" )
      wire#w1
      Contact( "Blend_T-40".Dose_Homomixer.QDOSERun )
      Contact( "Blend_T-40".Dose_Homomixer.P_CMD )
      wire#w2
      Coil( "T-14.00_Homomixer".IN_Dose_Pump_Cmd )
   END_RUNG
   RUNG wire#w1
      Contact( "Blend_T-41".Dose_Homomixer.QDOSERun )
      Contact( "Blend_T-41".Dose_Homomixer.P_CMD )
   END_RUNG wire#w2
   // the same network as SCL:
   "T-14.00_Homomixer".IN_Dose_Pump_Cmd := "AlwaysTRUE" AND (("Blend_T-40".Dose_Homomixer.QDOSERun AND "Blend_T-40".Dose_Homomixer.P_CMD) OR ("Blend_T-41".Dose_Homomixer.QDOSERun AND "Blend_T-41".Dose_Homomixer.P_CMD));
END_REGION

REGION Network 29: T-14.00 LineTransferOK
   RUNG wire#powerrail
      Contact( "AlwaysTRUE" )
      Contact( "T-14.00_Homomixer".IN_Dose_Run )
      wire#w1
      Contact( "Blend_T-40".IN_FBAV_Homomixer )
      wire#w2
      Coil( "T-14.00_Homomixer".IN_Dose_LineOK )
   END_RUNG
   RUNG wire#w1
      Contact( "Blend_T-41".IN_FBAV_Homomixer )
   END_RUNG wire#w2
   // the same network as SCL:
   "T-14.00_Homomixer".IN_Dose_LineOK := "AlwaysTRUE" AND "T-14.00_Homomixer".IN_Dose_Run AND ("Blend_T-40".IN_FBAV_Homomixer OR "Blend_T-41".IN_FBAV_Homomixer);
END_REGION

REGION Network 30: T-14.00 Homomixer
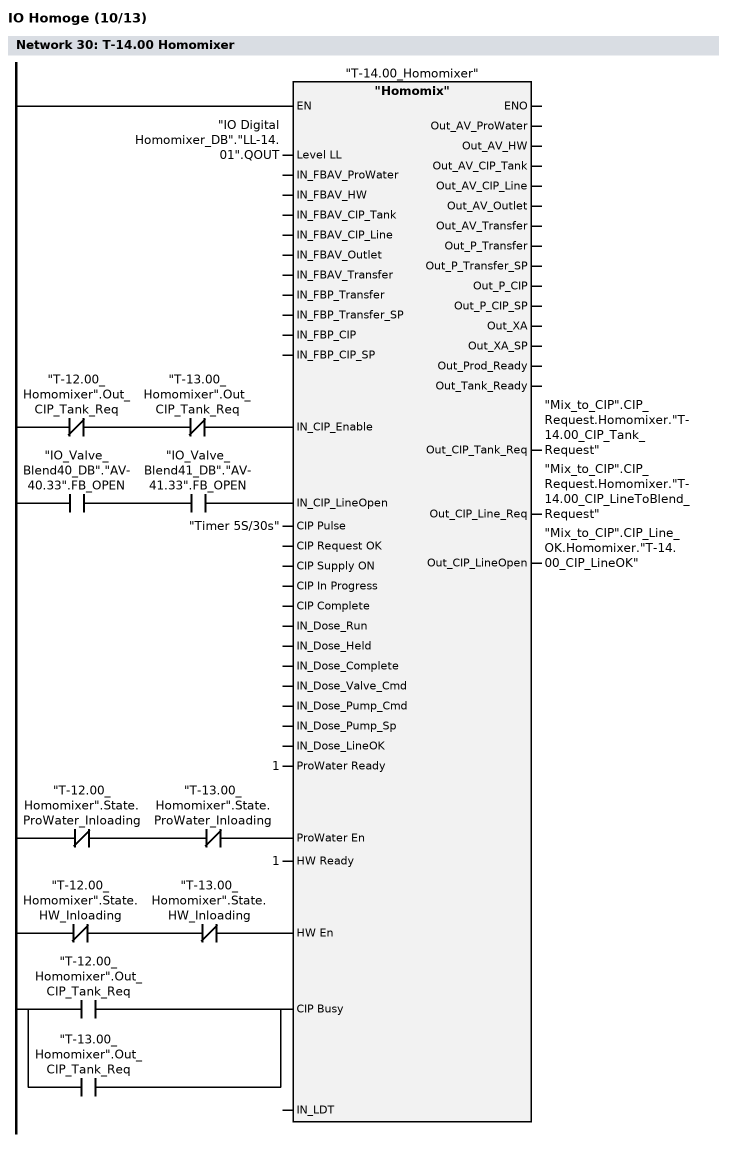
   RUNG wire#powerrail
      "T-14.00_Homomixer"(IN_CIP_Enable := wire#w1, IN_CIP_LineOpen := wire#w2, "ProWater En" := wire#w3, "HW En" := wire#w4, "CIP Busy" := wire#w5, "Level LL" := "IO Digital Homomixer_DB"."LL-14.01".QOUT, IN_FBAV_ProWater :=, IN_FBAV_HW :=, IN_FBAV_CIP_Tank :=, IN_FBAV_CIP_Line :=, IN_FBAV_Outlet :=, IN_FBAV_Transfer :=, IN_FBP_Transfer :=, IN_FBP_Transfer_SP :=, IN_FBP_CIP :=, IN_FBP_CIP_SP :=, "CIP Pulse" := "Timer 5S/30s", "CIP Request OK" :=, "CIP Supply ON" :=, "CIP In Progress" :=, "CIP Complete" :=, IN_Dose_Run :=, IN_Dose_Held :=, IN_Dose_Complete :=, IN_Dose_Valve_Cmd :=, IN_Dose_Pump_Cmd :=, IN_Dose_Pump_Sp :=, IN_Dose_LineOK :=, "ProWater Ready" := 1, "HW Ready" := 1, IN_LDT :=, Out_AV_ProWater =>, Out_AV_HW =>, Out_AV_CIP_Tank =>, Out_AV_CIP_Line =>, Out_AV_Outlet =>, Out_AV_Transfer =>, Out_P_Transfer =>, Out_P_Transfer_SP =>, Out_P_CIP =>, Out_P_CIP_SP =>, Out_XA =>, Out_XA_SP =>, Out_Prod_Ready =>, Out_Tank_Ready =>, Out_CIP_Tank_Req => "Mix_to_CIP".CIP_Request.Homomixer."T-14.00_CIP_Tank_Request", Out_CIP_Line_Req => "Mix_to_CIP".CIP_Request.Homomixer."T-14.00_CIP_LineToBlend_Request", Out_CIP_LineOpen => "Mix_to_CIP".CIP_Line_OK.Homomixer."T-14.00_CIP_LineOK")
   END_RUNG
   RUNG wire#powerrail
      I_Contact( "T-12.00_Homomixer".Out_CIP_Tank_Req )
      I_Contact( "T-13.00_Homomixer".Out_CIP_Tank_Req )
   END_RUNG wire#w1
   RUNG wire#powerrail
      Contact( "IO_Valve_Blend40_DB"."AV-40.33".FB_OPEN )
      Contact( "IO_Valve_Blend41_DB"."AV-41.33".FB_OPEN )
   END_RUNG wire#w2
   RUNG wire#powerrail
      I_Contact( "T-12.00_Homomixer".State.ProWater_Inloading )
      I_Contact( "T-13.00_Homomixer".State.ProWater_Inloading )
   END_RUNG wire#w3
   RUNG wire#powerrail
      I_Contact( "T-12.00_Homomixer".State.HW_Inloading )
      I_Contact( "T-13.00_Homomixer".State.HW_Inloading )
   END_RUNG wire#w4
   RUNG wire#powerrail
      Contact( "T-12.00_Homomixer".Out_CIP_Tank_Req )
   END_RUNG wire#w5
   RUNG wire#powerrail
      Contact( "T-13.00_Homomixer".Out_CIP_Tank_Req )
   END_RUNG wire#w5
   // the same network as SCL:
   "T-14.00_Homomixer"("Level LL" := "IO Digital Homomixer_DB"."LL-14.01".QOUT,   // "Homomix"
                       IN_CIP_Enable := NOT "T-12.00_Homomixer".Out_CIP_Tank_Req AND NOT "T-13.00_Homomixer".Out_CIP_Tank_Req,
                       IN_CIP_LineOpen := "IO_Valve_Blend40_DB"."AV-40.33".FB_OPEN AND "IO_Valve_Blend41_DB"."AV-41.33".FB_OPEN,
                       "CIP Pulse" := "Timer 5S/30s",
                       "ProWater Ready" := 1,
                       "ProWater En" := NOT "T-12.00_Homomixer".State.ProWater_Inloading AND NOT "T-13.00_Homomixer".State.ProWater_Inloading,
                       "HW Ready" := 1,
                       "HW En" := NOT "T-12.00_Homomixer".State.HW_Inloading AND NOT "T-13.00_Homomixer".State.HW_Inloading,
                       "CIP Busy" := "T-12.00_Homomixer".Out_CIP_Tank_Req OR "T-13.00_Homomixer".Out_CIP_Tank_Req,
                       Out_CIP_Tank_Req => "Mix_to_CIP".CIP_Request.Homomixer."T-14.00_CIP_Tank_Request",
                       Out_CIP_Line_Req => "Mix_to_CIP".CIP_Request.Homomixer."T-14.00_CIP_LineToBlend_Request",
                       Out_CIP_LineOpen => "Mix_to_CIP".CIP_Line_OK.Homomixer."T-14.00_CIP_LineOK");
END_REGION

REGION Network 31: T-14.00 Valve Cmd
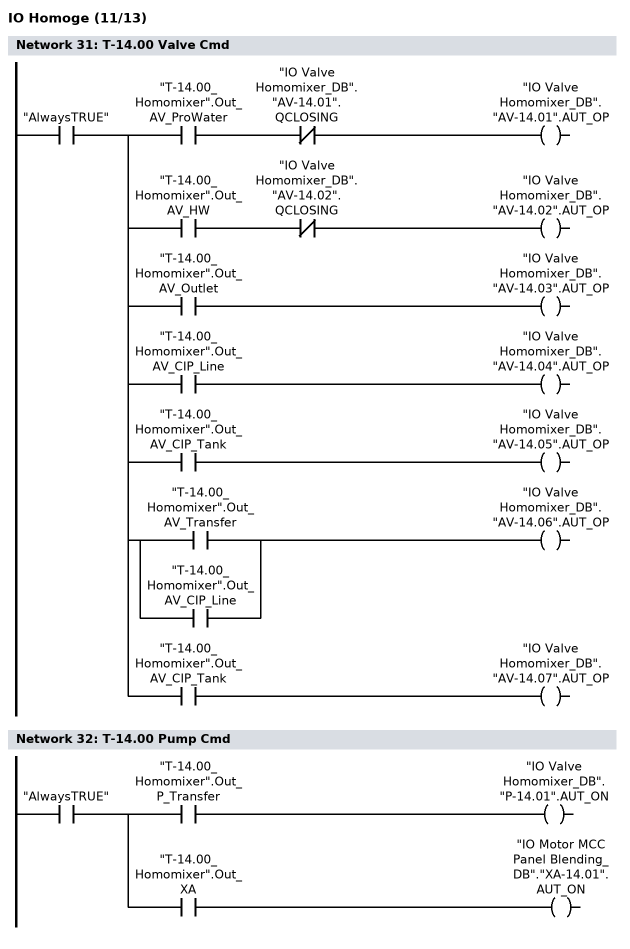
   RUNG wire#powerrail
      Contact( "AlwaysTRUE" )
      wire#w1
      Contact( "T-14.00_Homomixer".Out_AV_ProWater )
      I_Contact( "IO Valve Homomixer_DB"."AV-14.01".QCLOSING )
      Coil( "IO Valve Homomixer_DB"."AV-14.01".AUT_OP )
   END_RUNG
   RUNG wire#w1
      Contact( "T-14.00_Homomixer".Out_AV_HW )
      I_Contact( "IO Valve Homomixer_DB"."AV-14.02".QCLOSING )
      Coil( "IO Valve Homomixer_DB"."AV-14.02".AUT_OP )
   END_RUNG
   RUNG wire#w1
      Contact( "T-14.00_Homomixer".Out_AV_Outlet )
      Coil( "IO Valve Homomixer_DB"."AV-14.03".AUT_OP )
   END_RUNG
   RUNG wire#w1
      Contact( "T-14.00_Homomixer".Out_AV_CIP_Line )
      Coil( "IO Valve Homomixer_DB"."AV-14.04".AUT_OP )
   END_RUNG
   RUNG wire#w1
      Contact( "T-14.00_Homomixer".Out_AV_CIP_Tank )
      Coil( "IO Valve Homomixer_DB"."AV-14.05".AUT_OP )
   END_RUNG
   RUNG wire#w1
      Contact( "T-14.00_Homomixer".Out_AV_Transfer )
      wire#w2
      Coil( "IO Valve Homomixer_DB"."AV-14.06".AUT_OP )
   END_RUNG
   RUNG wire#w1
      Contact( "T-14.00_Homomixer".Out_AV_CIP_Line )
   END_RUNG wire#w2
   RUNG wire#w1
      Contact( "T-14.00_Homomixer".Out_AV_CIP_Tank )
      Coil( "IO Valve Homomixer_DB"."AV-14.07".AUT_OP )
   END_RUNG
   // the same network as SCL:
   "IO Valve Homomixer_DB"."AV-14.01".AUT_OP := "AlwaysTRUE" AND "T-14.00_Homomixer".Out_AV_ProWater AND NOT "IO Valve Homomixer_DB"."AV-14.01".QCLOSING;
   "IO Valve Homomixer_DB"."AV-14.02".AUT_OP := "AlwaysTRUE" AND "T-14.00_Homomixer".Out_AV_HW AND NOT "IO Valve Homomixer_DB"."AV-14.02".QCLOSING;
   "IO Valve Homomixer_DB"."AV-14.03".AUT_OP := "AlwaysTRUE" AND "T-14.00_Homomixer".Out_AV_Outlet;
   "IO Valve Homomixer_DB"."AV-14.04".AUT_OP := "AlwaysTRUE" AND "T-14.00_Homomixer".Out_AV_CIP_Line;
   "IO Valve Homomixer_DB"."AV-14.05".AUT_OP := "AlwaysTRUE" AND "T-14.00_Homomixer".Out_AV_CIP_Tank;
   "IO Valve Homomixer_DB"."AV-14.06".AUT_OP := "AlwaysTRUE" AND ("T-14.00_Homomixer".Out_AV_Transfer OR "T-14.00_Homomixer".Out_AV_CIP_Line);
   "IO Valve Homomixer_DB"."AV-14.07".AUT_OP := "AlwaysTRUE" AND "T-14.00_Homomixer".Out_AV_CIP_Tank;
END_REGION

REGION Network 32: T-14.00 Pump Cmd
   RUNG wire#powerrail
      Contact( "AlwaysTRUE" )
      wire#w1
      Contact( "T-14.00_Homomixer".Out_P_Transfer )
      Coil( "IO Valve Homomixer_DB"."P-14.01".AUT_ON )
   END_RUNG
   RUNG wire#w1
      Contact( "T-14.00_Homomixer".Out_XA )
      Coil( "IO Motor MCC Panel Blending_DB"."XA-14.01".AUT_ON )
   END_RUNG
   // the same network as SCL:
   "IO Valve Homomixer_DB"."P-14.01".AUT_ON := "AlwaysTRUE" AND "T-14.00_Homomixer".Out_P_Transfer;
   "IO Motor MCC Panel Blending_DB"."XA-14.01".AUT_ON := "AlwaysTRUE" AND "T-14.00_Homomixer".Out_XA;
END_REGION

REGION Network 33: T-14.00 Feedback Instrument
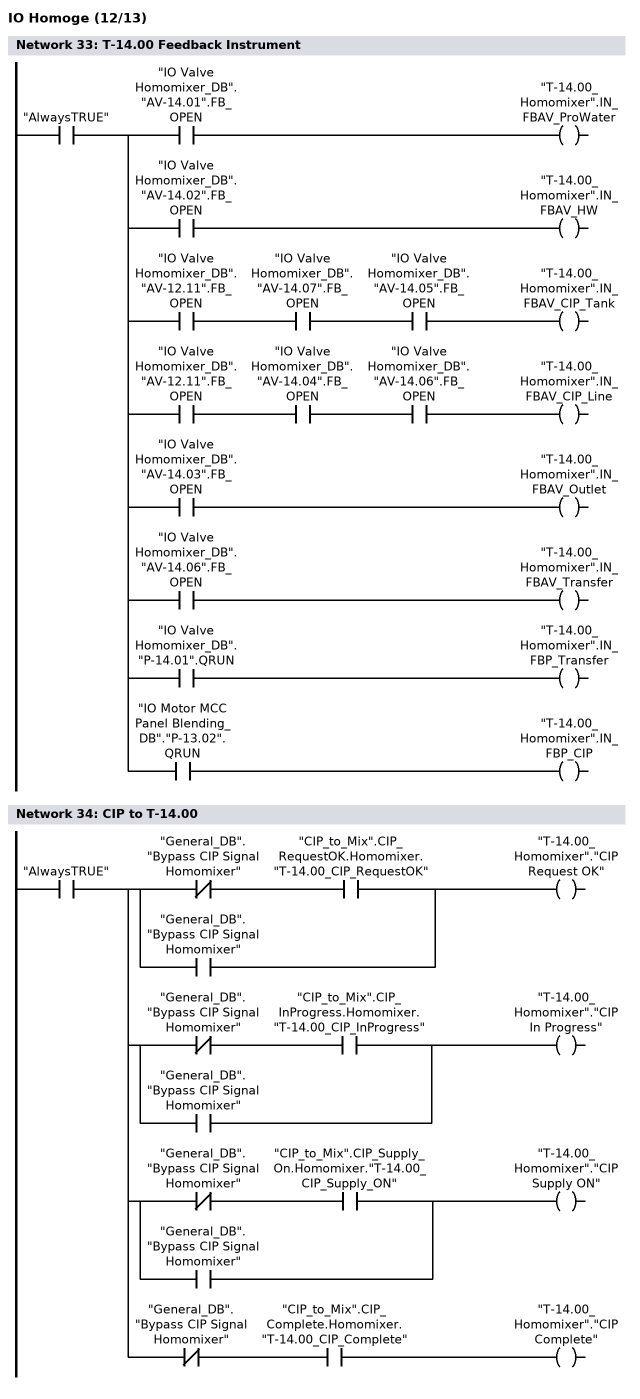
   RUNG wire#powerrail
      Contact( "AlwaysTRUE" )
      wire#w1
      Contact( "IO Valve Homomixer_DB"."AV-14.01".FB_OPEN )
      Coil( "T-14.00_Homomixer".IN_FBAV_ProWater )
   END_RUNG
   RUNG wire#w1
      Contact( "IO Valve Homomixer_DB"."AV-14.02".FB_OPEN )
      Coil( "T-14.00_Homomixer".IN_FBAV_HW )
   END_RUNG
   RUNG wire#w1
      Contact( "IO Valve Homomixer_DB"."AV-12.11".FB_OPEN )
      Contact( "IO Valve Homomixer_DB"."AV-14.07".FB_OPEN )
      Contact( "IO Valve Homomixer_DB"."AV-14.05".FB_OPEN )
      Coil( "T-14.00_Homomixer".IN_FBAV_CIP_Tank )
   END_RUNG
   RUNG wire#w1
      Contact( "IO Valve Homomixer_DB"."AV-12.11".FB_OPEN )
      Contact( "IO Valve Homomixer_DB"."AV-14.04".FB_OPEN )
      Contact( "IO Valve Homomixer_DB"."AV-14.06".FB_OPEN )
      Coil( "T-14.00_Homomixer".IN_FBAV_CIP_Line )
   END_RUNG
   RUNG wire#w1
      Contact( "IO Valve Homomixer_DB"."AV-14.03".FB_OPEN )
      Coil( "T-14.00_Homomixer".IN_FBAV_Outlet )
   END_RUNG
   RUNG wire#w1
      Contact( "IO Valve Homomixer_DB"."AV-14.06".FB_OPEN )
      Coil( "T-14.00_Homomixer".IN_FBAV_Transfer )
   END_RUNG
   RUNG wire#w1
      Contact( "IO Valve Homomixer_DB"."P-14.01".QRUN )
      Coil( "T-14.00_Homomixer".IN_FBP_Transfer )
   END_RUNG
   RUNG wire#w1
      Contact( "IO Motor MCC Panel Blending_DB"."P-13.02".QRUN )
      Coil( "T-14.00_Homomixer".IN_FBP_CIP )
   END_RUNG
   // the same network as SCL:
   "T-14.00_Homomixer".IN_FBAV_ProWater := "AlwaysTRUE" AND "IO Valve Homomixer_DB"."AV-14.01".FB_OPEN;
   "T-14.00_Homomixer".IN_FBAV_HW := "AlwaysTRUE" AND "IO Valve Homomixer_DB"."AV-14.02".FB_OPEN;
   "T-14.00_Homomixer".IN_FBAV_CIP_Tank := "AlwaysTRUE" AND "IO Valve Homomixer_DB"."AV-12.11".FB_OPEN AND "IO Valve Homomixer_DB"."AV-14.07".FB_OPEN AND "IO Valve Homomixer_DB"."AV-14.05".FB_OPEN;
   "T-14.00_Homomixer".IN_FBAV_CIP_Line := "AlwaysTRUE" AND "IO Valve Homomixer_DB"."AV-12.11".FB_OPEN AND "IO Valve Homomixer_DB"."AV-14.04".FB_OPEN AND "IO Valve Homomixer_DB"."AV-14.06".FB_OPEN;
   "T-14.00_Homomixer".IN_FBAV_Outlet := "AlwaysTRUE" AND "IO Valve Homomixer_DB"."AV-14.03".FB_OPEN;
   "T-14.00_Homomixer".IN_FBAV_Transfer := "AlwaysTRUE" AND "IO Valve Homomixer_DB"."AV-14.06".FB_OPEN;
   "T-14.00_Homomixer".IN_FBP_Transfer := "AlwaysTRUE" AND "IO Valve Homomixer_DB"."P-14.01".QRUN;
   "T-14.00_Homomixer".IN_FBP_CIP := "AlwaysTRUE" AND "IO Motor MCC Panel Blending_DB"."P-13.02".QRUN;
END_REGION

REGION Network 34: CIP to T-14.00
   RUNG wire#powerrail
      Contact( "AlwaysTRUE" )
      wire#w1
      I_Contact( "General_DB"."Bypass CIP Signal Homomixer" )
      Contact( "CIP_to_Mix".CIP_RequestOK.Homomixer."T-14.00_CIP_RequestOK" )
      wire#w2
      Coil( "T-14.00_Homomixer"."CIP Request OK" )
   END_RUNG
   RUNG wire#w1
      Contact( "General_DB"."Bypass CIP Signal Homomixer" )
   END_RUNG wire#w2
   RUNG wire#w1
      I_Contact( "General_DB"."Bypass CIP Signal Homomixer" )
      Contact( "CIP_to_Mix".CIP_InProgress.Homomixer."T-14.00_CIP_InProgress" )
      wire#w3
      Coil( "T-14.00_Homomixer"."CIP In Progress" )
   END_RUNG
   RUNG wire#w1
      Contact( "General_DB"."Bypass CIP Signal Homomixer" )
   END_RUNG wire#w3
   RUNG wire#w1
      I_Contact( "General_DB"."Bypass CIP Signal Homomixer" )
      Contact( "CIP_to_Mix".CIP_Supply_On.Homomixer."T-14.00_CIP_Supply_ON" )
      wire#w4
      Coil( "T-14.00_Homomixer"."CIP Supply ON" )
   END_RUNG
   RUNG wire#w1
      Contact( "General_DB"."Bypass CIP Signal Homomixer" )
   END_RUNG wire#w4
   RUNG wire#w1
      I_Contact( "General_DB"."Bypass CIP Signal Homomixer" )
      Contact( "CIP_to_Mix".CIP_Complete.Homomixer."T-14.00_CIP_Complete" )
      Coil( "T-14.00_Homomixer"."CIP Complete" )
   END_RUNG
   // the same network as SCL:
   "T-14.00_Homomixer"."CIP Request OK" := "AlwaysTRUE" AND ((NOT "General_DB"."Bypass CIP Signal Homomixer" AND "CIP_to_Mix".CIP_RequestOK.Homomixer."T-14.00_CIP_RequestOK") OR "General_DB"."Bypass CIP Signal Homomixer");
   "T-14.00_Homomixer"."CIP In Progress" := "AlwaysTRUE" AND ((NOT "General_DB"."Bypass CIP Signal Homomixer" AND "CIP_to_Mix".CIP_InProgress.Homomixer."T-14.00_CIP_InProgress") OR "General_DB"."Bypass CIP Signal Homomixer");
   "T-14.00_Homomixer"."CIP Supply ON" := "AlwaysTRUE" AND ((NOT "General_DB"."Bypass CIP Signal Homomixer" AND "CIP_to_Mix".CIP_Supply_On.Homomixer."T-14.00_CIP_Supply_ON") OR "General_DB"."Bypass CIP Signal Homomixer");
   "T-14.00_Homomixer"."CIP Complete" := "AlwaysTRUE" AND NOT "General_DB"."Bypass CIP Signal Homomixer" AND "CIP_to_Mix".CIP_Complete.Homomixer."T-14.00_CIP_Complete";
END_REGION

REGION Network 36: Valve CIP Supply AV-12.11
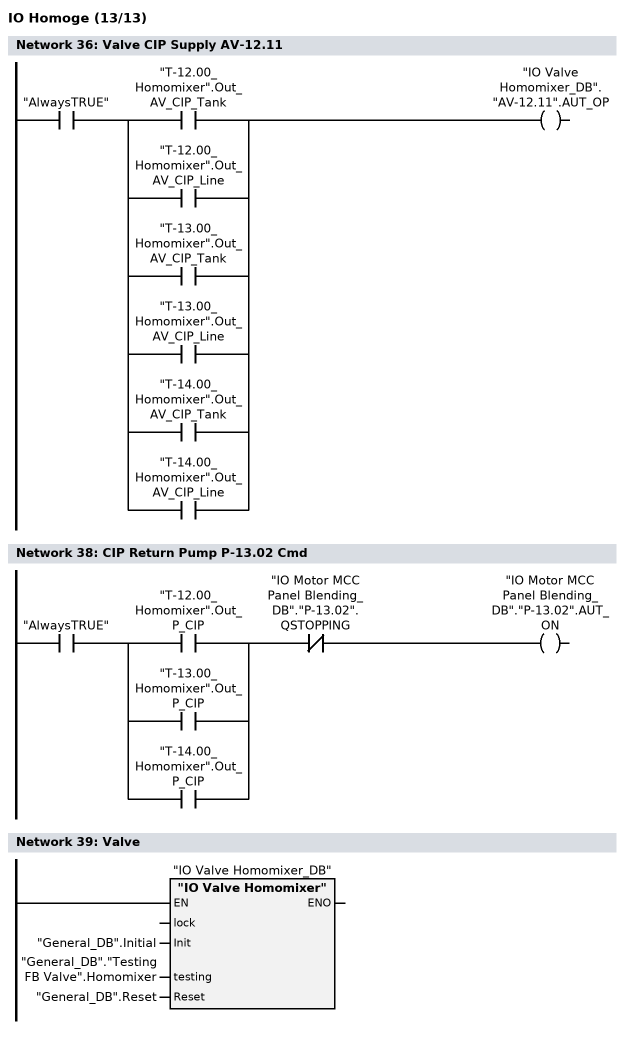
   RUNG wire#powerrail
      Contact( "AlwaysTRUE" )
      wire#w1
      Contact( "T-12.00_Homomixer".Out_AV_CIP_Tank )
      wire#w2
      Coil( "IO Valve Homomixer_DB"."AV-12.11".AUT_OP )
   END_RUNG
   RUNG wire#w1
      Contact( "T-12.00_Homomixer".Out_AV_CIP_Line )
   END_RUNG wire#w2
   RUNG wire#w1
      Contact( "T-13.00_Homomixer".Out_AV_CIP_Tank )
   END_RUNG wire#w2
   RUNG wire#w1
      Contact( "T-13.00_Homomixer".Out_AV_CIP_Line )
   END_RUNG wire#w2
   RUNG wire#w1
      Contact( "T-14.00_Homomixer".Out_AV_CIP_Tank )
   END_RUNG wire#w2
   RUNG wire#w1
      Contact( "T-14.00_Homomixer".Out_AV_CIP_Line )
   END_RUNG wire#w2
   // the same network as SCL:
   "IO Valve Homomixer_DB"."AV-12.11".AUT_OP := "AlwaysTRUE" AND ("T-12.00_Homomixer".Out_AV_CIP_Tank OR "T-12.00_Homomixer".Out_AV_CIP_Line OR "T-13.00_Homomixer".Out_AV_CIP_Tank OR "T-13.00_Homomixer".Out_AV_CIP_Line OR "T-14.00_Homomixer".Out_AV_CIP_Tank OR "T-14.00_Homomixer".Out_AV_CIP_Line);
END_REGION

REGION Network 37: Valve Drain AV-12.12 for T-12 T-13 T-14
END_REGION

REGION Network 38: CIP Return Pump P-13.02 Cmd
   RUNG wire#powerrail
      Contact( "AlwaysTRUE" )
      wire#w1
      Contact( "T-12.00_Homomixer".Out_P_CIP )
      wire#w2
      I_Contact( "IO Motor MCC Panel Blending_DB"."P-13.02".QSTOPPING )
      Coil( "IO Motor MCC Panel Blending_DB"."P-13.02".AUT_ON )
   END_RUNG
   RUNG wire#w1
      Contact( "T-13.00_Homomixer".Out_P_CIP )
   END_RUNG wire#w2
   RUNG wire#w1
      Contact( "T-14.00_Homomixer".Out_P_CIP )
   END_RUNG wire#w2
   // the same network as SCL:
   "IO Motor MCC Panel Blending_DB"."P-13.02".AUT_ON := "AlwaysTRUE" AND ("T-12.00_Homomixer".Out_P_CIP OR "T-13.00_Homomixer".Out_P_CIP OR "T-14.00_Homomixer".Out_P_CIP) AND NOT "IO Motor MCC Panel Blending_DB"."P-13.02".QSTOPPING;
END_REGION

REGION Network 39: Valve
   RUNG wire#powerrail
      "IO Valve Homomixer_DB"(lock :=, Init := "General_DB".Initial, testing := "General_DB"."Testing FB Valve".Homomixer, Reset := "General_DB".Reset)
   END_RUNG
   // the same network as SCL:
   "IO Valve Homomixer_DB"(Init := "General_DB".Initial,   // "IO Valve Homomixer"
                           testing := "General_DB"."Testing FB Valve".Homomixer,
                           Reset := "General_DB".Reset);
END_REGION
END_FUNCTION
